// Mitsubishi GX Works2 project: PLC_Final_0804   PLC: FX3G

// global labels: Global1
VAR_GLOBAL
  ActiveWork AT Y007 : BOOL;
  StartWorkdaySwitch AT X007 : BOOL;
END_VAR
VAR_GLOBAL CONSTANT
  Chocolate : REAL := 1200;
END_VAR
VAR_GLOBAL
  ChocolateInventory AT D1100 : REAL;
END_VAR
VAR_GLOBAL CONSTANT
  Nuts : REAL := 300;
END_VAR
VAR_GLOBAL
  NutsInventory AT D1200 : REAL;
END_VAR
VAR_GLOBAL CONSTANT
  Pistachio : REAL := 300;
END_VAR
VAR_GLOBAL
  PistachioInventory AT D1300 : REAL;
END_VAR
VAR_GLOBAL CONSTANT
  Kadayif : REAL := 120;
END_VAR
VAR_GLOBAL
  KadayifInventory AT D1400 : REAL;
  BreakWorkdaySwitch AT X005 : BOOL;
END_VAR
VAR_GLOBAL CONSTANT
  ChocolateMin : REAL := 400;
  NutsMin : REAL := 100;
  PistachioMin : REAL := 120;
  KadayifMin : REAL := 60;
END_VAR
VAR_GLOBAL
  ActiveMelting AT Y001 : BOOL;
  StartMeltingSwitch AT X001 : BOOL;
  StartDayIndication AT M0 : BOOL;
  EndDayIndication AT M1 : BOOL;
  MeltingContainer AT D1500 : REAL;
  TempSensor AT X002 : BOOL;
  CastingTimer AT TS10 : BOOL;
  StartCastingIndication AT M2 : BOOL;
  ProximitySensor AT X003 : BOOL;
  Templates AT D1600 : REAL;
  ActiveCasting AT M3 : BOOL;
  EndMeltingIndication AT M2 : BOOL;
  CastingProcess AT Y002 : BOOL;
  CastingrCoil AT TC10 : BOOL;
END_VAR
VAR_GLOBAL CONSTANT
  CastingDuration : INT := 40;
END_VAR
VAR_GLOBAL
  EndCastingIndication AT M4 : BOOL;
  SampleInputSwitch AT X004 : BOOL;
  AnalogInput1 AT D8280 : INT;
  SampleValue AT D1700 : REAL;
END_VAR
VAR_GLOBAL CONSTANT
  NutsThreshold : REAL := 5;
END_VAR
VAR_GLOBAL
  NutsProductionIndicator AT M5 : BOOL;
END_VAR
VAR_GLOBAL CONSTANT
  NutsRequiredForNutsMix : REAL := 100;
END_VAR
VAR_GLOBAL
  NutsMixProductionIndicator AT M5 : BOOL;
END_VAR
VAR_GLOBAL CONSTANT
  NutsMixThreshold : REAL := 5;
  PistachioRequiredForNutsMix : REAL := 100;
END_VAR
VAR_GLOBAL
  FillingCreamContainer AT D1800 : REAL;
END_VAR
VAR_GLOBAL CONSTANT
  NutsRequiredForDubai : REAL := 20;
  PistachioRequiredForDubai : REAL := 120;
  KadayifRequiredForDubai : REAL := 60;
END_VAR
VAR_GLOBAL
  StartFillingIndicator AT M6 : BOOL;
END_VAR
VAR_GLOBAL CONSTANT
  CreamFillingDuration : WORD := 50;
END_VAR
VAR_GLOBAL
  CreamFillingCoil AT TC20 : BOOL;
  FillingTimer AT TS20 : BOOL;
  Flash2 AT Y004 : BOOL;
  Flash1Coil AT TC30 : BOOL;
END_VAR
VAR_GLOBAL CONSTANT
  BlinkingTime : WORD := 5;
END_VAR
VAR_GLOBAL
  Flash1Timer AT TS30 : BOOL;
  Flash1 AT Y003 : BOOL;
  Flash2Coil AT TC40 : BOOL;
  Flash2Timer AT TS40 : BOOL;
  DubaiProductionIndicator AT M7 : BOOL;
END_VAR
VAR_GLOBAL CONSTANT
  DivConstant : REAL := 400;
END_VAR
VAR_GLOBAL
  CoolingTimer AT TS50 : BOOL;
  EndFillingIndications AT M8 : BOOL;
  EndFillingIndication AT M8 : BOOL;
  CoolingSwitch AT X006 : BOOL;
  CoolingProcess AT Y006 : BOOL;
  CoolingCoil AT TC50 : BOOL;
END_VAR
VAR_GLOBAL CONSTANT
  CoolingDuration : INT := 30;
END_VAR
VAR_GLOBAL
  StartCoolingProcess AT M9 : BOOL;
  PackingCounter AT CS1 : BOOL;
  EndCoolingIndication AT M10 : BOOL;
  PackChocolateSwitch AT X000 : BOOL;
END_VAR
VAR_GLOBAL CONSTANT
  AmountPerPackage : WORD := 4;
END_VAR
VAR_GLOBAL
  PackingCounterCoil AT CC1 : BOOL;
  ActivePacking AT Y005 : BOOL;
  UnitsContainer AT D1900 : REAL;
END_VAR
VAR_GLOBAL CONSTANT
  UnitIncrement : REAL := 1;
END_VAR
VAR_GLOBAL
  StartPackingIndication AT M11 : BOOL;
  AnalogOutput AT D8282 : INT;
END_VAR
VAR_GLOBAL CONSTANT
  MultiplyConstant : REAL := 40;
  RegistersRange : WORD := K801;
  ResetValue : REAL;
  ResetValueOutput : WORD;
END_VAR
VAR_GLOBAL
  ChocolateShortageIndicator AT M12 : BOOL;
END_VAR
VAR_GLOBAL CONSTANT
  CreamAmount : REAL := 200;
END_VAR
VAR_GLOBAL
  ActiveWorkdayIndication AT M0 : BOOL;
  InventoryShortageIndication AT M1 : BOOL;
  EmergencySwitch AT X005 : BOOL;
  CastingCoil AT TC10 : BOOL;
END_VAR

// task Task_01 (event TRUE, interval 0, priority 31): POU_01

PROGRAM POU_01
(* structured ladder/FBD written out as ST: instructions are called as NAME(EN, inputs, outputs); _pN, _eN, _tN stand for wires *)
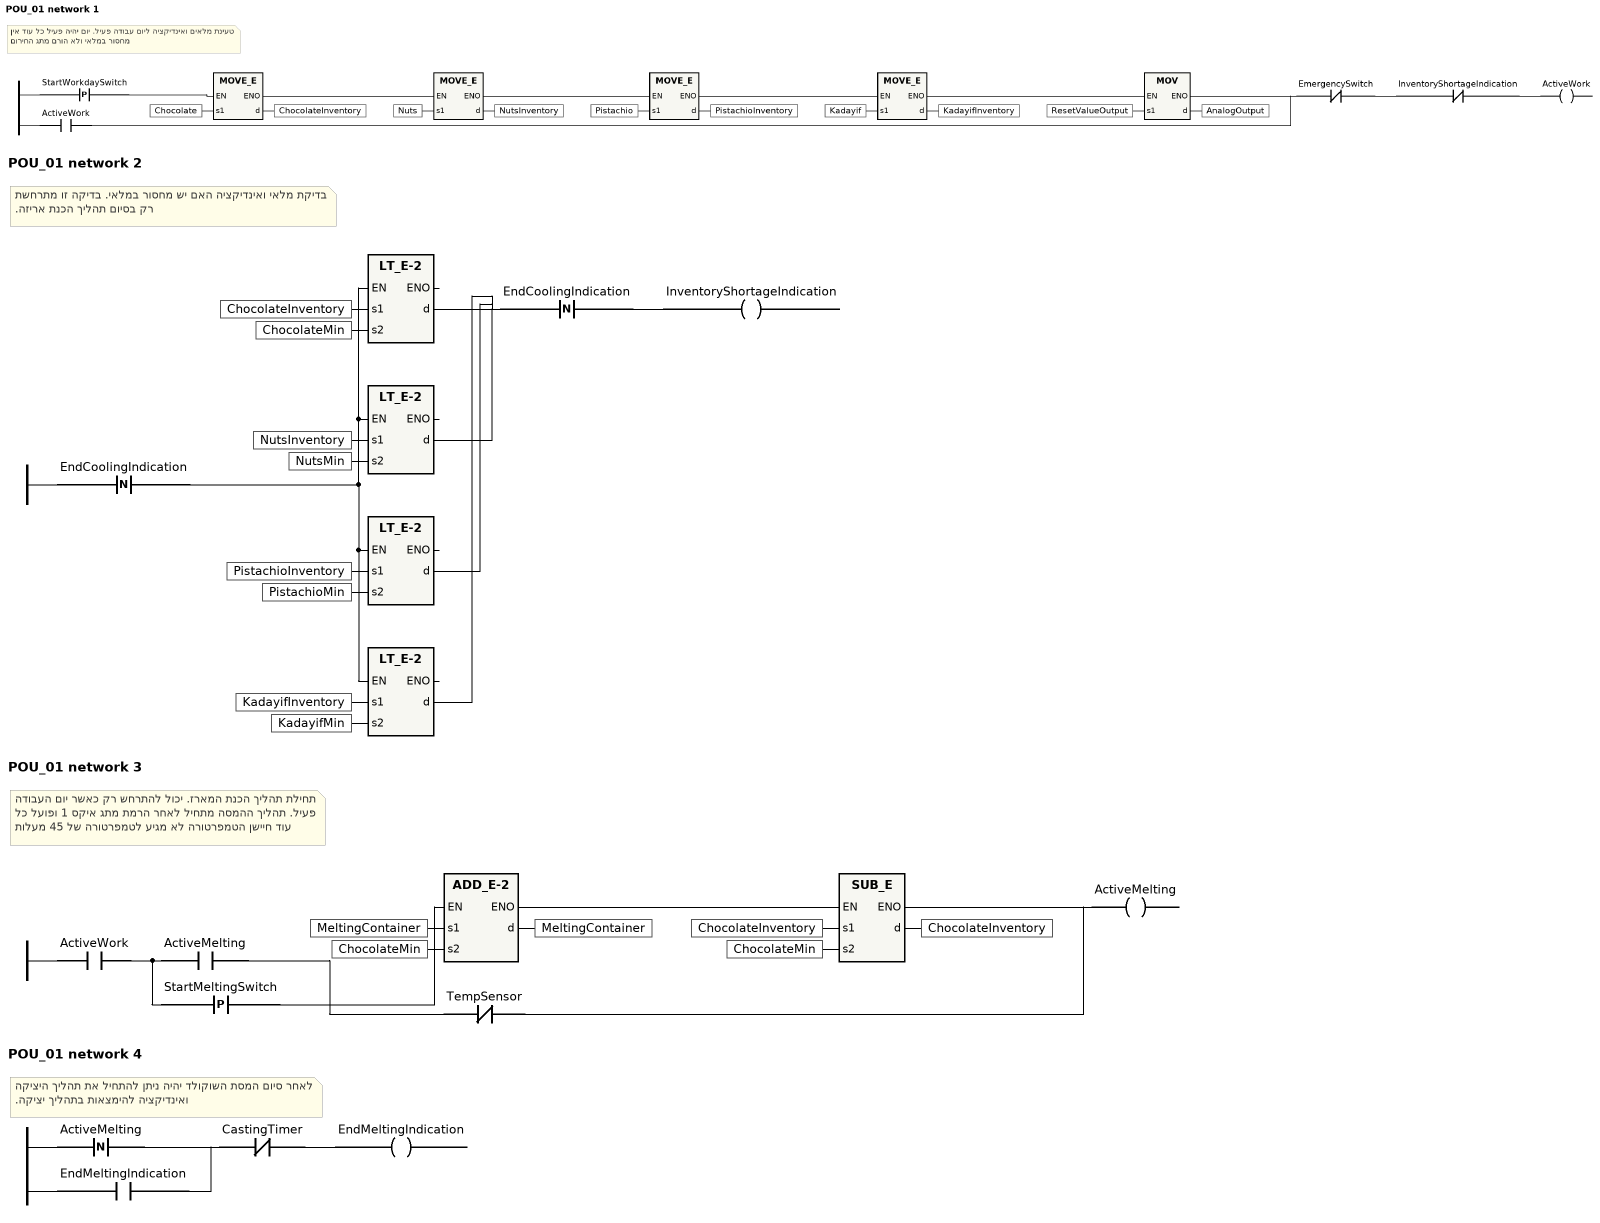
(* network 1 *)
(* טעינת מלאים ואינדיקציה ליום עבודה פעיל. יום יהיה פעיל כל עוד אין מחסור במלאי ולא הורם מתג החירום *)
_e1 := MOVE_E(LDP(TRUE, StartWorkdaySwitch), Chocolate, ChocolateInventory);
_e2 := MOVE_E(_e1, Nuts, NutsInventory);
_e3 := MOVE_E(_e2, Pistachio, PistachioInventory);
_e4 := MOVE_E(_e3, Kadayif, KadayifInventory);
_e5 := MOV(_e4, ResetValueOutput, AnalogOutput);
ActiveWork := ((_e5 OR ActiveWork) AND NOT EmergencySwitch) AND NOT InventoryShortageIndication;
(* network 2 *)
(* בדיקת מלאי ואינדיקציה האם יש מחסור במלאי. בדיקה זו מתרחשת רק בסיום תהליך הכנת אריזה. *)
_p1 := LDF(TRUE, EndCoolingIndication);
LT_E(_p1, ChocolateInventory, ChocolateMin, _t2);
LT_E(_p1, NutsInventory, NutsMin, _t3);
LT_E(_p1, PistachioInventory, PistachioMin, _t4);
LT_E(_p1, KadayifInventory, KadayifMin, _t5);
InventoryShortageIndication := (_t2 OR _t3 OR _t4 OR _t5) AND LDF(TRUE, EndCoolingIndication);
(* network 3 *)
(* תחילת תהליך הכנת המארז. יכול להתרחש רק כאשר יום העבודה פעיל. תהליך ההמסה מתחיל לאחר הרמת מתג איקס 1 ופועל כל עוד חיישן הטמפרטורה לא מגיע לטמפרטורה של 45 מעלות *)
_e1 := ADD_E(ActiveWork AND LDP(TRUE, StartMeltingSwitch), MeltingContainer, ChocolateMin, MeltingContainer);
_e2 := SUB_E(_e1, ChocolateInventory, ChocolateMin, ChocolateInventory);
ActiveMelting := (ActiveWork AND ActiveMelting AND NOT TempSensor) OR _e2;
(* network 4 *)
(* לאחר סיום המסת השוקולד יהיה ניתן להתחיל את תהליך היציקה ואינדיקציה להימצאות בתהליך יציקה. *)
EndMeltingIndication := (LDF(TRUE, ActiveMelting) OR EndMeltingIndication) AND NOT CastingTimer;
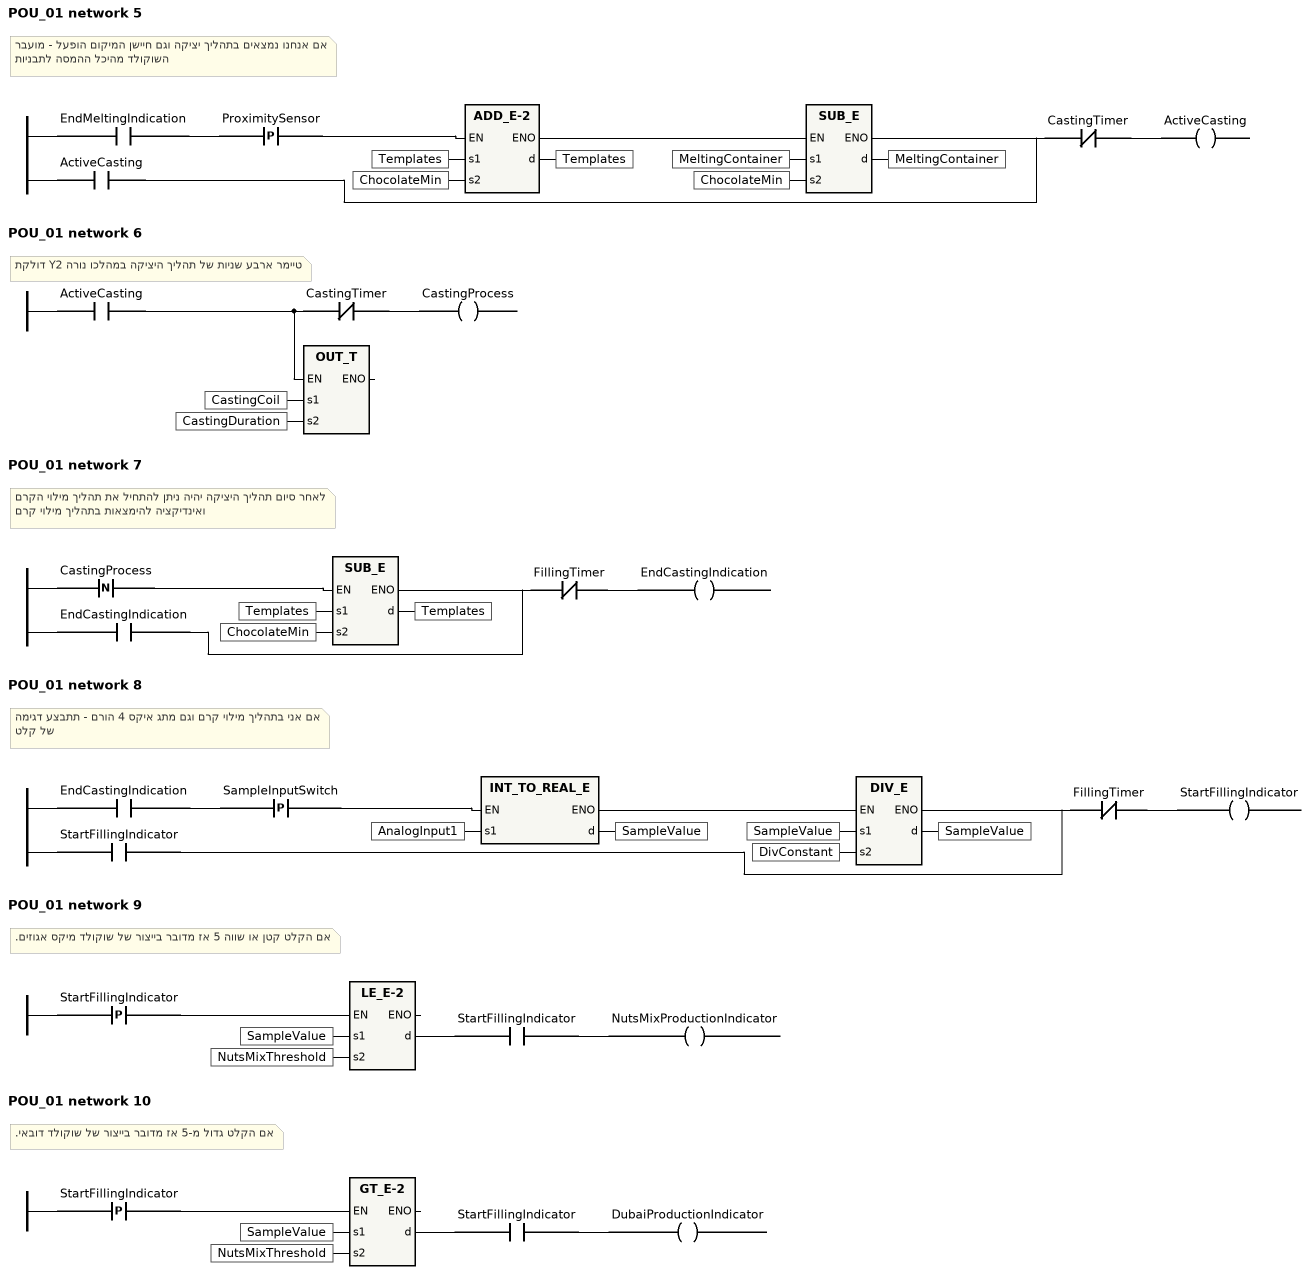
(* network 5 *)
(* אם אנחנו נמצאים בתהליך יציקה וגם חיישן המיקום הופעל - מועבר השוקולד מהיכל ההמסה לתבניות *)
_e1 := ADD_E(EndMeltingIndication AND LDP(TRUE, ProximitySensor), Templates, ChocolateMin, Templates);
_e2 := SUB_E(_e1, MeltingContainer, ChocolateMin, MeltingContainer);
ActiveCasting := (_e2 OR ActiveCasting) AND NOT CastingTimer;
(* network 6 *)
(* טיימר ארבע שניות של תהליך היציקה במהלכו נורה Y2 דולקת *)
CastingProcess := ActiveCasting AND NOT CastingTimer;
OUT_T(ActiveCasting, CastingCoil, CastingDuration);
(* network 7 *)
(* לאחר סיום תהליך היציקה יהיה ניתן להתחיל את תהליך מילוי הקרם ואינדיקציה להימצאות בתהליך מילוי קרם *)
_e1 := SUB_E(LDF(TRUE, CastingProcess), Templates, ChocolateMin, Templates);
EndCastingIndication := (_e1 OR EndCastingIndication) AND NOT FillingTimer;
(* network 8 *)
(* אם אני בתהליך מילוי קרם וגם מתג איקס 4 הורם - תתבצע דגימה של קלט *)
_e1 := INT_TO_REAL_E(EndCastingIndication AND LDP(TRUE, SampleInputSwitch), AnalogInput1, SampleValue);
_e2 := DIV_E(_e1, SampleValue, DivConstant, SampleValue);
StartFillingIndicator := (_e2 OR StartFillingIndicator) AND NOT FillingTimer;
(* network 9 *)
(* אם הקלט קטן או שווה 5 אז מדובר בייצור של שוקולד מיקס אגוזים. *)
LE_E(LDP(TRUE, StartFillingIndicator), SampleValue, NutsMixThreshold, _t1);
NutsMixProductionIndicator := _t1 AND StartFillingIndicator;
(* network 10 *)
(* אם הקלט גדול מ-5 אז מדובר בייצור של שוקולד דובאי. *)
GT_E(LDP(TRUE, StartFillingIndicator), SampleValue, NutsMixThreshold, _t1);
DubaiProductionIndicator := _t1 AND StartFillingIndicator;
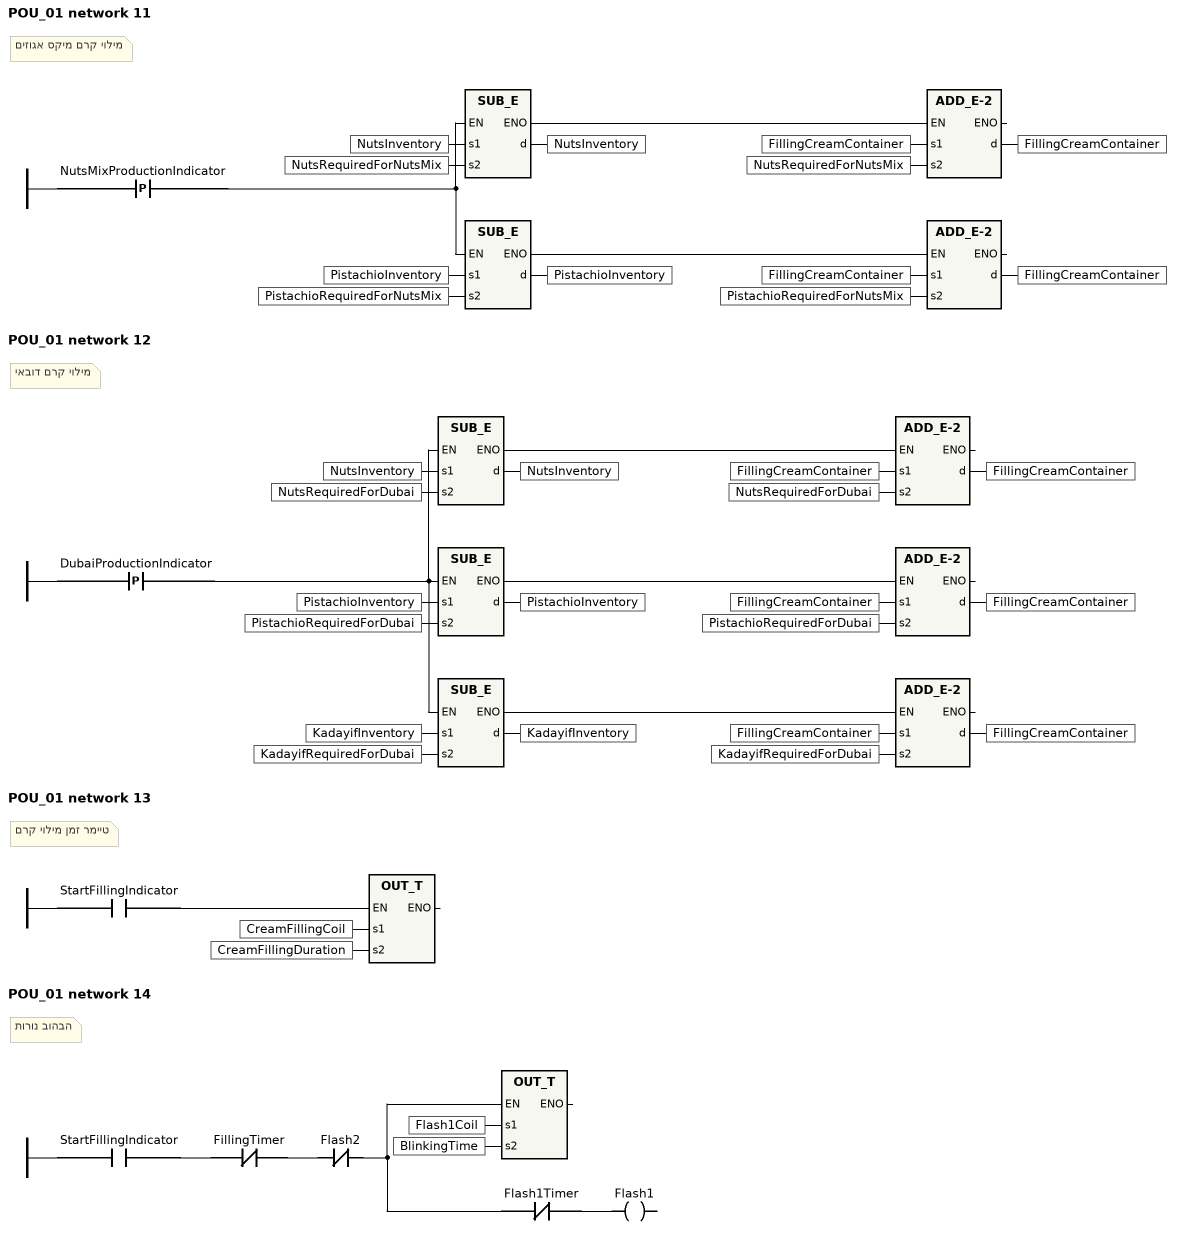
(* network 11 *)
(* מילוי קרם מיקס אגוזים *)
_p1 := LDP(TRUE, NutsMixProductionIndicator);
_e2 := SUB_E(_p1, NutsInventory, NutsRequiredForNutsMix, NutsInventory);
ADD_E(_e2, FillingCreamContainer, NutsRequiredForNutsMix, FillingCreamContainer);
_e3 := SUB_E(_p1, PistachioInventory, PistachioRequiredForNutsMix, PistachioInventory);
ADD_E(_e3, FillingCreamContainer, PistachioRequiredForNutsMix, FillingCreamContainer);
(* network 12 *)
(* מילוי קרם דובאי *)
_p1 := LDP(TRUE, DubaiProductionIndicator);
_e2 := SUB_E(_p1, NutsInventory, NutsRequiredForDubai, NutsInventory);
ADD_E(_e2, FillingCreamContainer, NutsRequiredForDubai, FillingCreamContainer);
_e3 := SUB_E(_p1, PistachioInventory, PistachioRequiredForDubai, PistachioInventory);
ADD_E(_e3, FillingCreamContainer, PistachioRequiredForDubai, FillingCreamContainer);
_e4 := SUB_E(_p1, KadayifInventory, KadayifRequiredForDubai, KadayifInventory);
ADD_E(_e4, FillingCreamContainer, KadayifRequiredForDubai, FillingCreamContainer);
(* network 13 *)
(* טיימר זמן מילוי קרם *)
OUT_T(StartFillingIndicator, CreamFillingCoil, CreamFillingDuration);
(* network 14 *)
(* הבהוב נורות *)
_p1 := StartFillingIndicator AND NOT FillingTimer AND NOT Flash2;
OUT_T(_p1, Flash1Coil, BlinkingTime);
Flash1 := _p1 AND NOT Flash1Timer;
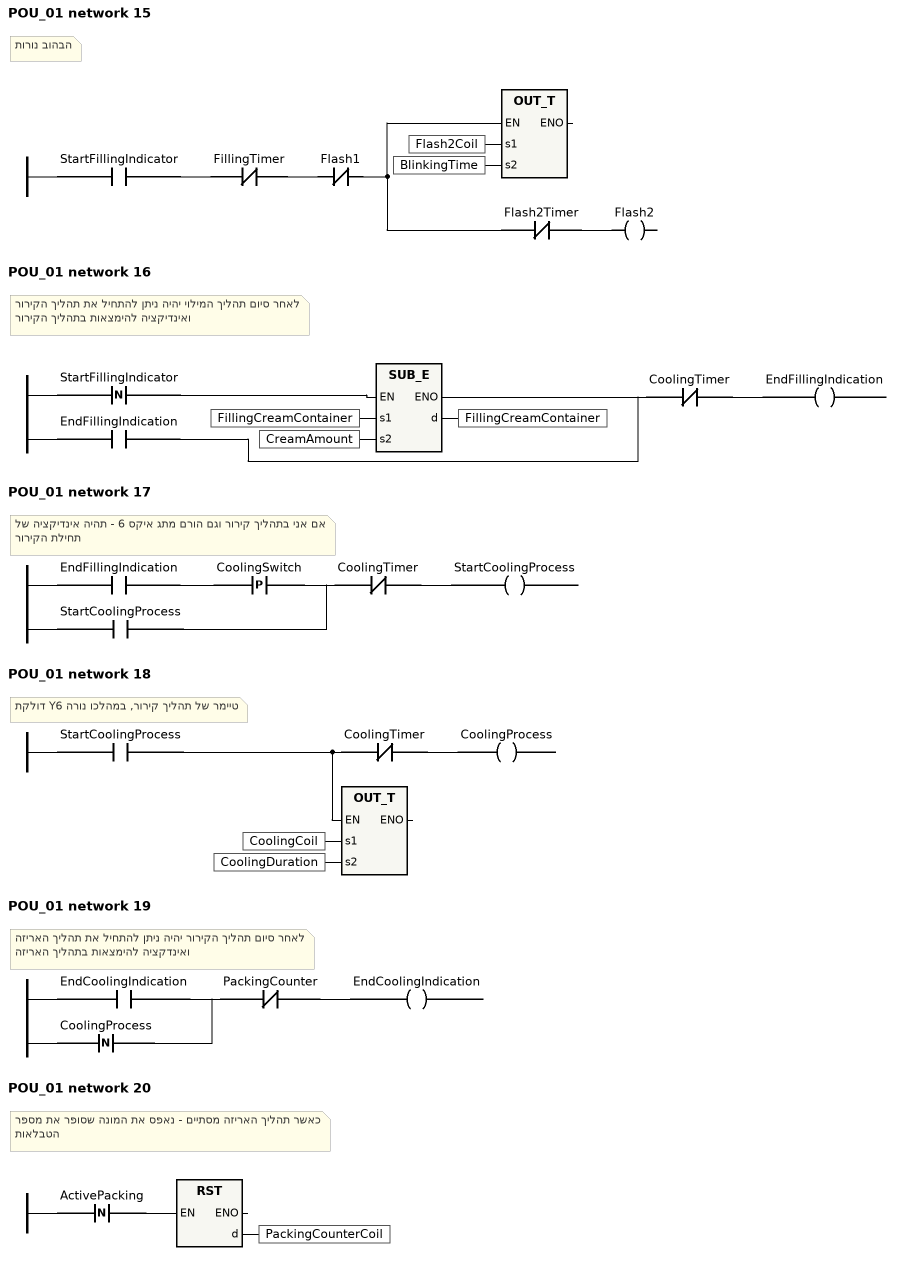
(* network 15 *)
(* הבהוב נורות *)
_p1 := StartFillingIndicator AND NOT FillingTimer AND NOT Flash1;
OUT_T(_p1, Flash2Coil, BlinkingTime);
Flash2 := _p1 AND NOT Flash2Timer;
(* network 16 *)
(* לאחר סיום תהליך המילוי יהיה ניתן להתחיל את תהליך הקירור ואינדיקציה להימצאות בתהליך הקירור *)
_e1 := SUB_E(LDF(TRUE, StartFillingIndicator), FillingCreamContainer, CreamAmount, FillingCreamContainer);
EndFillingIndication := (_e1 OR EndFillingIndication) AND NOT CoolingTimer;
(* network 17 *)
(* אם אני בתהליך קירור וגם הורם מתג איקס 6 - תהיה אינדיקציה של תחילת הקירור *)
StartCoolingProcess := ((EndFillingIndication AND LDP(TRUE, CoolingSwitch)) OR StartCoolingProcess) AND NOT CoolingTimer;
(* network 18 *)
(* טיימר של תהליך קירור, במהלכו נורה Y6 דולקת *)
CoolingProcess := StartCoolingProcess AND NOT CoolingTimer;
OUT_T(StartCoolingProcess, CoolingCoil, CoolingDuration);
(* network 19 *)
(* לאחר סיום תהליך הקירור יהיה ניתן להתחיל את תהליך האריזה ואינדקציה להימצאות בתהליך האריזה *)
EndCoolingIndication := (EndCoolingIndication OR LDF(TRUE, CoolingProcess)) AND NOT PackingCounter;
(* network 20 *)
(* כאשר תהליך האריזה מסתיים - נאפס את המונה שסופר את מספר הטבלאות *)
RST(LDF(TRUE, ActivePacking), PackingCounterCoil);
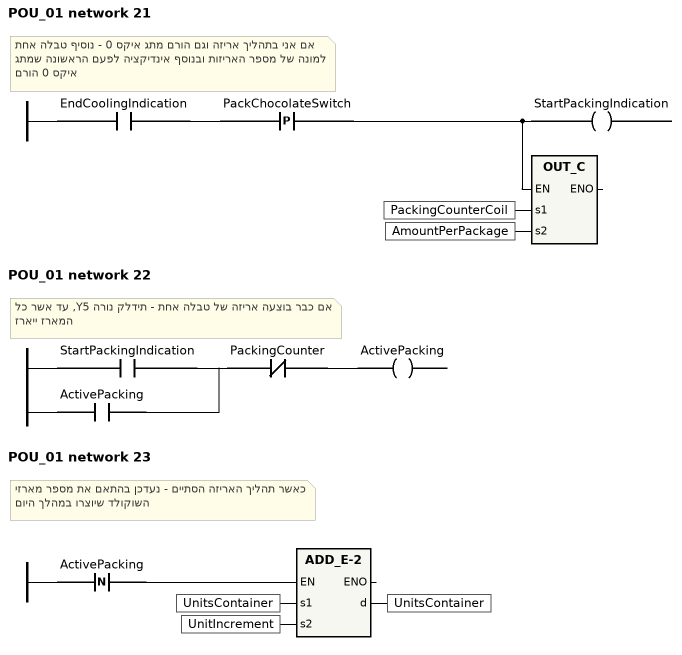
(* network 21 *)
(* אם אני בתהליך אריזה וגם הורם מתג איקס 0 - נוסיף טבלה אחת למונה של מספר האריזות ובנוסף אינדיקציה לפעם הראשונה שמתג איקס 0 הורם *)
_p1 := EndCoolingIndication AND LDP(TRUE, PackChocolateSwitch);
StartPackingIndication := _p1;
OUT_C(_p1, PackingCounterCoil, AmountPerPackage);
(* network 22 *)
(* אם כבר בוצעה אריזה של טבלה אחת - תידלק נורה Y5, עד אשר כל המארז ייארז *)
ActivePacking := (StartPackingIndication OR ActivePacking) AND NOT PackingCounter;
(* network 23 *)
(* כאשר תהליך האריזה הסתיים - נעדכן בהתאם את מספר מארזי השוקולד שיוצרו במהלך היום *)
ADD_E(LDF(TRUE, ActivePacking), UnitsContainer, UnitIncrement, UnitsContainer);
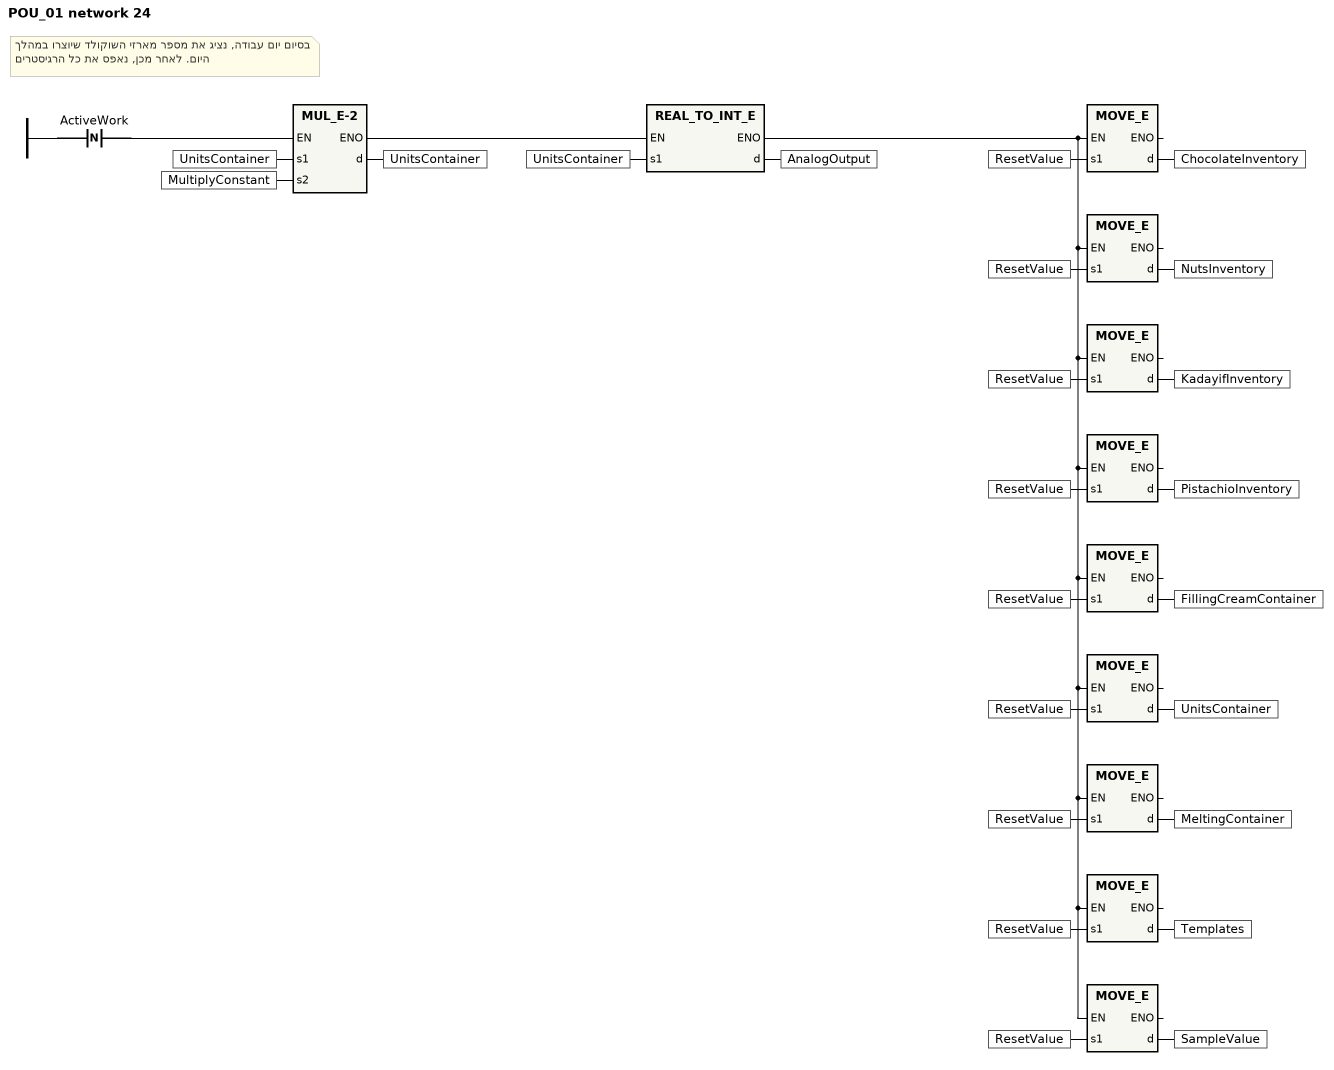
(* network 24 *)
(* בסיום יום עבודה, נציג את מספר מארזי השוקולד שיוצרו במהלך היום. לאחר מכן, נאפס את כל הרגיסטרים *)
_e1 := MUL_E(LDF(TRUE, ActiveWork), UnitsContainer, MultiplyConstant, UnitsContainer);
_e2 := REAL_TO_INT_E(_e1, UnitsContainer, AnalogOutput);
MOVE_E(_e2, ResetValue, ChocolateInventory);
MOVE_E(_e2, ResetValue, NutsInventory);
MOVE_E(_e2, ResetValue, KadayifInventory);
MOVE_E(_e2, ResetValue, PistachioInventory);
MOVE_E(_e2, ResetValue, FillingCreamContainer);
MOVE_E(_e2, ResetValue, UnitsContainer);
MOVE_E(_e2, ResetValue, MeltingContainer);
MOVE_E(_e2, ResetValue, Templates);
MOVE_E(_e2, ResetValue, SampleValue);
END_PROGRAM
